(* IEC 61131-3 sources: ST-Study/patterns, 3 files *)

(* ---- fb_alarm_manager.st ---- *)
(*
===============================================================================
  报警管理模块 - FB_AlarmManager
===============================================================================
  功能: 管理多路报警,支持锁存/复位/确认/消抖/优先级
  作者: ST 学习系统
  版本: v1.0
  日期: 2025-12-21

  使用场景:
  - 管理多个报警源(传感器故障、超时、越限等)
  - 需要报警锁存(故障瞬间消失也要记录)
  - 需要报警确认(操作员必须确认才能消除)
  - 需要报警消抖(避免抖动误报)

  核心功能:
  1. 报警锁存: 触发后即使条件消失也保持
  2. 报警复位: 需要人工确认或自动复位
  3. 报警消抖: 信号稳定一段时间才触发
  4. 优先级分类: 严重/警告/提示

  接口说明(单路报警版):
  输入:
    iAlarmTrigger   : BOOL  - 报警触发条件
    iReset          : BOOL  - 复位信号
    iAutoReset      : BOOL  - 允许自动复位
    tDebounceTime   : TIME  - 消抖时间
    nPriority       : INT   - 优先级(1=提示,2=警告,3=严重)

  输出:
    oAlarmActive    : BOOL  - 报警有效(锁存后)
    oAlarmRaw       : BOOL  - 原始报警(消抖后,未锁存)
    oAlarmNew       : BOOL  - 新报警(上升沿脉冲)

  使用示例:
    fbAlarm_MotorOverload(
        iAlarmTrigger := MotorCurrent > MAX_CURRENT,
        iReset := ResetButton,
        iAutoReset := FALSE,  // 严重故障,必须人工复位
        tDebounceTime := T#500ms,
        nPriority := 3,
        oAlarmActive => AlarmLamp
    );
===============================================================================
*)

FUNCTION_BLOCK FB_Alarm
(*
    单路报警模块(基础版)
*)
VAR_INPUT
    iAlarmTrigger   : BOOL;         // 报警触发条件
    iReset          : BOOL;         // 复位信号
    iAutoReset      : BOOL;         // 允许自动复位
    tDebounceTime   : TIME := T#0s; // 消抖时间(0表示不消抖)
    nPriority       : INT := 2;     // 优先级(1=提示,2=警告,3=严重)
END_VAR

VAR_OUTPUT
    oAlarmActive    : BOOL;         // 报警有效(锁存后)
    oAlarmRaw       : BOOL;         // 原始报警(消抖后)
    oAlarmNew       : BOOL;         // 新报警标志(上升沿)
END_VAR

VAR
    fbDebounce      : TON;          // 消抖定时器
    bAlarmLatched   : BOOL;         // 报警锁存
    rtAlarm         : R_TRIG;       // 报警上升沿
    rtReset         : R_TRIG;       // 复位上升沿
END_VAR

// === 消抖处理 ===
fbDebounce(IN := iAlarmTrigger, PT := tDebounceTime);

IF tDebounceTime > T#0s THEN
    oAlarmRaw := fbDebounce.Q;  // 有消抖时间,使用定时器输出
ELSE
    oAlarmRaw := iAlarmTrigger; // 无消抖时间,直接使用原始信号
END_IF

// === 报警锁存 ===
rtAlarm(CLK := oAlarmRaw);
IF rtAlarm.Q THEN
    bAlarmLatched := TRUE;  // 上升沿锁存
END_IF

// === 报警复位 ===
rtReset(CLK := iReset);

// 人工复位
IF rtReset.Q THEN
    bAlarmLatched := FALSE;
END_IF

// 自动复位(条件消失且允许自动复位)
IF iAutoReset AND NOT oAlarmRaw THEN
    bAlarmLatched := FALSE;
END_IF

// === 输出赋值 ===
oAlarmActive := bAlarmLatched;
oAlarmNew := rtAlarm.Q;  // 新报警脉冲(用于计数/记录)

END_FUNCTION_BLOCK

(*
===============================================================================
  多路报警管理器 - FB_AlarmManager
===============================================================================
  管理多路报警(最多16路)
  提供统一的复位、优先级排序、报警计数功能
===============================================================================
*)

FUNCTION_BLOCK FB_AlarmManager

VAR_INPUT
    iAlarmTriggers  : ARRAY[1..16] OF BOOL;  // 16路报警触发条件
    iResetAll       : BOOL;                   // 全部复位
    iResetSingle    : INT;                    // 单路复位(1-16, 0=无)
END_VAR

VAR_OUTPUT
    oAlarmActive    : ARRAY[1..16] OF BOOL;  // 16路报警状态
    oAnyAlarm       : BOOL;                   // 任意报警有效
    oAlarmCount     : INT;                    // 当前报警数量
    oHighestPriority: INT;                    // 最高优先级(3=严重,2=警告,1=提示)
END_VAR

VAR
    fbAlarms        : ARRAY[1..16] OF FB_Alarm;  // 16个报警实例
    i               : INT;                        // 循环变量

    // 每路报警的配置(可外部配置或在此硬编码)
    aPriority       : ARRAY[1..16] OF INT := [
        3, 3, 2, 2, 2, 2, 1, 1,  // 路1-8
        1, 1, 1, 1, 1, 1, 1, 1   // 路9-16
    ];

    aDebounceTime   : ARRAY[1..16] OF TIME := [
        T#500ms, T#500ms, T#300ms, T#300ms, T#300ms, T#300ms, T#200ms, T#200ms,
        T#200ms, T#200ms, T#200ms, T#200ms, T#200ms, T#200ms, T#200ms, T#200ms
    ];

    aAutoReset      : ARRAY[1..16] OF BOOL := [
        FALSE, FALSE, FALSE, FALSE, TRUE, TRUE, TRUE, TRUE,
        TRUE, TRUE, TRUE, TRUE, TRUE, TRUE, TRUE, TRUE
    ];
END_VAR

// === 循环处理每路报警 ===
oAlarmCount := 0;
oHighestPriority := 0;

FOR i := 1 TO 16 DO
    // 调用单路报警模块
    fbAlarms[i](
        iAlarmTrigger := iAlarmTriggers[i],
        iReset := iResetAll OR (iResetSingle = i),
        iAutoReset := aAutoReset[i],
        tDebounceTime := aDebounceTime[i],
        nPriority := aPriority[i],
        oAlarmActive => oAlarmActive[i]
    );

    // 统计报警数量
    IF oAlarmActive[i] THEN
        oAlarmCount := oAlarmCount + 1;

        // 更新最高优先级
        IF aPriority[i] > oHighestPriority THEN
            oHighestPriority := aPriority[i];
        END_IF
    END_IF
END_FOR

// === 任意报警标志 ===
oAnyAlarm := (oAlarmCount > 0);

END_FUNCTION_BLOCK

(*
===============================================================================
  使用示例1: 单路报警
===============================================================================

VAR
    fbAlarm_MotorOverload : FB_Alarm;
    MotorCurrent : REAL;
    MAX_CURRENT : REAL := 10.0;
END_VAR

// 电机过载报警
fbAlarm_MotorOverload(
    iAlarmTrigger := (MotorCurrent > MAX_CURRENT),  // 触发条件
    iReset := HMI.ResetButton,                       // 复位按钮
    iAutoReset := FALSE,                             // 必须人工复位
    tDebounceTime := T#500ms,                        // 消抖500ms
    nPriority := 3,                                  // 严重报警
    oAlarmActive => HMI.AlarmLamp                    // 输出到报警灯
);

// 报警触发时停机
IF fbAlarm_MotorOverload.oAlarmActive THEN
    Motor.iStop := TRUE;
END_IF

===============================================================================
  使用示例2: 多路报警管理
===============================================================================

VAR
    fbAlarmMgr : FB_AlarmManager;

    // 报警触发条件
    bOverload : BOOL;
    bOverheat : BOOL;
    bLowPressure : BOOL;
    // ...
END_VAR

// 配置报警触发条件
fbAlarmMgr.iAlarmTriggers[1] := bOverload;       // 路1: 过载
fbAlarmMgr.iAlarmTriggers[2] := bOverheat;       // 路2: 过热
fbAlarmMgr.iAlarmTriggers[3] := bLowPressure;    // 路3: 低压
// ...

// 调用报警管理器
fbAlarmMgr(
    iResetAll := HMI.ResetAllButton,
    iResetSingle := HMI.SelectedAlarmIndex  // 单个复位
);

// 显示报警状态
HMI.AlarmCount := fbAlarmMgr.oAlarmCount;
HMI.AnyAlarmActive := fbAlarmMgr.oAnyAlarm;

// 根据优先级控制报警灯颜色
CASE fbAlarmMgr.oHighestPriority OF
    3: HMI.AlarmLampColor := RED;     // 严重
    2: HMI.AlarmLampColor := YELLOW;  // 警告
    1: HMI.AlarmLampColor := BLUE;    // 提示
    ELSE
        HMI.AlarmLampColor := OFF;
END_CASE

===============================================================================
  使用示例3: 报警与状态机联动
===============================================================================

FUNCTION_BLOCK FB_MachineControl
VAR
    fbAlarmMgr : FB_AlarmManager;
    nState : INT;
END_VAR

// 严重报警时自动停机
IF fbAlarmMgr.oHighestPriority >= 3 THEN
    nState := STATE_ERROR;  // 进入错误状态
END_IF

// 警告时仅提示,不停机
IF fbAlarmMgr.oHighestPriority = 2 THEN
    HMI.WarningMessage := 'Warning: Check system';
END_IF

END_FUNCTION_BLOCK

===============================================================================
  测试清单
===============================================================================

【基础功能】
1. 触发条件成立 → oAlarmActive=TRUE
2. 触发条件消失,人工复位 → oAlarmActive=FALSE

【锁存机制】
3. 触发条件瞬间成立(100ms)后消失 → oAlarmActive=TRUE(锁存保持)
4. 锁存后必须复位才能消除 → 即使触发条件消失也保持

【消抖功能】
5. 触发条件抖动(ON 100ms, OFF 100ms) → 无报警(未达到消抖时间)
6. 触发条件稳定500ms → 报警触发

【自动复位】
7. 允许自动复位,触发条件消失 → oAlarmActive=FALSE(自动复位)
8. 不允许自动复位,触发条件消失 → oAlarmActive=TRUE(保持,需人工复位)

【多路报警】
9. 3路同时报警 → oAlarmCount=3, oAnyAlarm=TRUE
10. 复位全部 → oAlarmCount=0, oAnyAlarm=FALSE
11. 单个复位路2 → 路2复位,其他保持

【优先级排序】
12. 路1(严重),路3(警告)同时报警 → oHighestPriority=3
13. 路1复位后 → oHighestPriority=2

【边界条件】
14. 连续触发10次 → oAlarmNew只在第一次触发时为TRUE(上升沿)
15. 复位按钮连按10次 → 只复位一次(边沿检测)

===============================================================================
  设计要点
===============================================================================

1. **锁存 vs 非锁存**:
   - 锁存: 故障瞬间即记录,需人工确认(适用于严重故障)
   - 非锁存(自动复位): 条件消失即恢复(适用于轻微提示)

2. **消抖时间选择**:
   - 机械触点: 50-200ms
   - 传感器信号: 100-500ms
   - 模拟量越限: 500-1000ms(避免边界抖动)

3. **优先级分类建议**:
   - 3 严重: 必须立即停机(过载、急停、安全门打开)
   - 2 警告: 需要关注但可继续运行(温度偏高、压力偏低)
   - 1 提示: 仅提示信息(维护提醒、计数达到)

4. **报警历史记录**(扩展):
   - 可添加 ARRAY[1..100] OF AlarmRecord 记录最近100条
   - 记录: 时间戳、报警ID、触发值、复位时间

5. **报警优先级显示**:
   - 严重: 红色闪烁 + 蜂鸣器
   - 警告: 黄色常亮
   - 提示: 蓝色常亮

===============================================================================
*)

(* ---- fb_pause_resume.st ---- *)
(*
===============================================================================
  全局暂停保持模块 - FB_PauseResume
===============================================================================
  功能: 提供全局暂停保持功能,支持多设备同步暂停/恢复
  作者: ST 学习系统
  版本: v1.0
  日期: 2025-12-21

  使用场景:
  - 整条生产线的全局暂停(所有设备同步暂停)
  - 需要保持现场状态的暂停(不是急停,而是"定格")
  - 需要从暂停点精确恢复的场景

  核心思想:
  - 暂停时"冻结"所有状态,不改变任何输出
  - 恢复时从冻结点继续,不重复执行已完成的动作
  - 提供"暂停允许条件"检查,避免危险位置暂停

  接口说明:
  输入:
    iPauseRequest   : BOOL  - 暂停请求
    iResumeRequest  : BOOL  - 恢复请求
    iEmergencyStop  : BOOL  - 急停(强制暂停,不检查条件)
    iPauseEnable    : BOOL  - 暂停允许条件(TRUE时才能暂停)

  输出:
    oPaused         : BOOL  - 当前已暂停
    oPauseActive    : BOOL  - 暂停信号有效(供其他模块读取)
    oResuming       : BOOL  - 恢复中(可用于渐进恢复)
    oPauseRejected  : BOOL  - 暂停请求被拒绝(条件不满足)

  使用示例:
    // 1. 在主程序中实例化(全局单例)
    fbGlobalPause : FB_PauseResume;

    // 2. 调用
    fbGlobalPause(
        iPauseRequest := PauseButton,
        iResumeRequest := ResumeButton,
        iEmergencyStop := EmergencyStop,
        iPauseEnable := SafePositionReached,  // 只在安全位置允许暂停
        oPaused => SystemPaused,
        oPauseActive => GlobalPauseSignal
    );

    // 3. 其他模块响应暂停信号
    IF fbGlobalPause.oPauseActive THEN
        // 冻结当前状态,不改变输出
        RETURN;  // 提前退出,不执行后续逻辑
    END_IF
===============================================================================
*)

FUNCTION_BLOCK FB_PauseResume

VAR_INPUT
    iPauseRequest   : BOOL;     // 暂停请求
    iResumeRequest  : BOOL;     // 恢复请求
    iEmergencyStop  : BOOL;     // 急停信号
    iPauseEnable    : BOOL;     // 暂停允许条件
END_VAR

VAR_OUTPUT
    oPaused         : BOOL;     // 当前已暂停
    oPauseActive    : BOOL;     // 暂停信号有效(供其他模块读取)
    oResuming       : BOOL;     // 恢复中
    oPauseRejected  : BOOL;     // 暂停请求被拒绝
END_VAR

VAR
    bPausedState    : BOOL;     // 暂停状态锁存
    bResumingState  : BOOL;     // 恢复状态

    rtPause         : R_TRIG;   // 暂停上升沿
    rtResume        : R_TRIG;   // 恢复上升沿

    fbRejectPulse   : TP;       // 拒绝脉冲(用于显示)

    CONST_REJECT_PULSE_TIME : TIME := T#2s;  // 拒绝提示持续时间
END_VAR

// === 边沿检测 ===
rtPause(CLK := iPauseRequest);
rtResume(CLK := iResumeRequest);

// === 暂停逻辑 ===
IF rtPause.Q THEN
    // 检查暂停条件
    IF iPauseEnable OR iEmergencyStop THEN
        // 条件满足,执行暂停
        bPausedState := TRUE;
        bResumingState := FALSE;
        oPauseRejected := FALSE;
    ELSE
        // 条件不满足,拒绝暂停
        fbRejectPulse(IN := TRUE, PT := CONST_REJECT_PULSE_TIME);
    END_IF
END_IF

// === 急停强制暂停(优先级最高) ===
IF iEmergencyStop THEN
    bPausedState := TRUE;
    bResumingState := FALSE;
END_IF

// === 恢复逻辑 ===
IF rtResume.Q AND bPausedState AND NOT iEmergencyStop THEN
    bPausedState := FALSE;
    bResumingState := TRUE;  // 进入恢复中状态
END_IF

// === 恢复中状态处理(可用于渐进恢复) ===
IF bResumingState THEN
    // 这里可以添加渐进恢复逻辑
    // 例如:先恢复低速,再恢复正常速度
    // 目前简化为立即恢复
    bResumingState := FALSE;
END_IF

// === 输出赋值 ===
oPaused := bPausedState;
oPauseActive := bPausedState;  // 供其他模块读取的暂停信号
oResuming := bResumingState;

// === 拒绝提示脉冲 ===
fbRejectPulse(IN := FALSE);  // 自动关闭输入
oPauseRejected := fbRejectPulse.Q;

END_FUNCTION_BLOCK

(*
===============================================================================
  使用模式1: 全局暂停(单例模式)
===============================================================================

// === 在全局变量(GVL)中声明 ===
VAR_GLOBAL
    fbGlobalPause : FB_PauseResume;  // 全局唯一实例
END_VAR

// === 在主程序中调用 ===
PROGRAM Main
VAR
    SafePositionReached : BOOL;  // 安全位置标志
END_VAR

// 调用全局暂停模块
fbGlobalPause(
    iPauseRequest := HMI.PauseButton,
    iResumeRequest := HMI.ResumeButton,
    iEmergencyStop := IO.EmergencyStop,
    iPauseEnable := SafePositionReached,  // 只在安全位置允许暂停
    oPaused => HMI.PausedLamp,
    oPauseRejected => HMI.PauseRejectedAlarm
);

// 检查安全位置(示例:所有电机都停止)
SafePositionReached :=
    NOT Motor1.oRunning AND
    NOT Motor2.oRunning AND
    NOT Conveyor.oRunning;

END_PROGRAM

===============================================================================
  使用模式2: 状态机响应全局暂停
===============================================================================

FUNCTION_BLOCK FB_ConveyorControl
VAR_INPUT
    iStart : BOOL;
END_VAR
VAR_OUTPUT
    oRunning : BOOL;
END_VAR
VAR
    nState : INT;
END_VAR

// === 暂停优先检查(在状态机最前面) ===
IF fbGlobalPause.oPauseActive THEN
    // 暂停时冻结状态,不执行后续逻辑
    RETURN;
END_IF

// === 状态机正常逻辑 ===
CASE nState OF
    0: // 空闲
        IF iStart THEN
            nState := 10;
        END_IF

    10: // 启动
        oRunning := TRUE;
        // ...
END_CASE

END_FUNCTION_BLOCK

===============================================================================
  使用模式3: 渐进恢复(高级用法)
===============================================================================

// 修改 FB_PauseResume 的恢复逻辑:
VAR
    fbResumeDelay : TON;  // 恢复延时
    nResumePhase : INT;   // 恢复阶段
END_VAR

// 恢复时分阶段处理
IF rtResume.Q AND bPausedState AND NOT iEmergencyStop THEN
    bPausedState := FALSE;
    bResumingState := TRUE;
    nResumePhase := 1;  // 开始第一阶段
END_IF

IF bResumingState THEN
    CASE nResumePhase OF
        1:  // 第一阶段:低速恢复
            fbResumeDelay(IN := TRUE, PT := T#2s);
            IF fbResumeDelay.Q THEN
                nResumePhase := 2;
                fbResumeDelay(IN := FALSE);
            END_IF

        2:  // 第二阶段:正常速度
            bResumingState := FALSE;
            nResumePhase := 0;
    END_CASE
END_IF

// 其他模块根据 oResuming 调整速度
IF fbGlobalPause.oResuming THEN
    MotorSpeed := LowSpeed;  // 恢复阶段使用低速
ELSE
    MotorSpeed := NormalSpeed;
END_IF

===============================================================================
  测试清单
===============================================================================

【基础功能】
1. 按暂停按钮(条件满足) → oPaused=TRUE, 所有设备冻结
2. 暂停状态按恢复 → oPaused=FALSE, 设备从暂停点继续

【暂停条件检查】
3. 设备运行中按暂停(条件不满足) → oPauseRejected=TRUE, 暂停失败
4. 设备停止后按暂停(条件满足) → oPaused=TRUE, 暂停成功

【急停处理】
5. 运行中急停 → oPaused=TRUE (强制暂停,不检查条件)
6. 急停状态按恢复 → 无效,必须先解除急停

【状态保持】
7. 暂停时传送带位置X → 恢复后仍从位置X继续(不回退)
8. 暂停时计数器值100 → 恢复后从100继续计数(不清零)

【边界条件】
9. 连续按暂停10次 → 只暂停一次(边沿检测)
10. 暂停后立即按恢复 → 正常恢复(无延时限制)
11. 未暂停时按恢复 → 无效(无副作用)

【多设备同步】
12. 3台电机运行,暂停 → 3台同时冻结
13. 恢复 → 3台同时恢复,保持相对位置关系

【拒绝提示】
14. 暂停被拒绝 → oPauseRejected 保持2秒(提示用户)

===============================================================================
  设计要点
===============================================================================

1. **暂停 ≠ 急停**:
   - 暂停: 可控的、可恢复的、保持现场的"定格"
   - 急停: 紧急的、安全的、可能丢失状态的"硬停"

2. **暂停条件检查**:
   - 避免危险位置暂停(如:机械手在空中)
   - 建议: 只在设备停稳、无运动时允许暂停
   - 特殊需求: 可以设计"运动中暂停"(需要额外的位置保存逻辑)

3. **状态冻结技巧**:
   - 在每个FB最前面检查 oPauseActive
   - 如果暂停,RETURN 提前退出,不执行后续逻辑
   - 不改变任何输出,保持现场

4. **恢复策略**:
   - 简单场景: 直接恢复
   - 复杂场景: 渐进恢复(低速→正常速度)
   - 安全场景: 恢复前重新检查安全条件

5. **全局单例模式**:
   - 整个系统只需要一个 FB_PauseResume 实例
   - 在全局变量(GVL)中声明
   - 所有模块读取同一个 oPauseActive 信号

===============================================================================
*)

(* ---- fb_state_machine.st ---- *)
(*
===============================================================================
  通用状态机框架 - FB_StateMachine
===============================================================================
  功能: 提供标准的状态机结构,支持暂停保持/恢复/异常回退
  作者: ST 学习系统
  版本: v1.0
  日期: 2025-12-21

  使用场景:
  - 任何需要步进控制的场景(传送带启动、机械手动作、工序流程等)
  - 需要暂停保持和恢复续跑的自动化流程
  - 需要异常处理和安全回退的控制逻辑

  接口说明:
  输入:
    iStart      : BOOL  - 启动信号(上升沿触发)
    iReset      : BOOL  - 复位信号(回到初始状态)
    iPause      : BOOL  - 暂停信号(保持当前状态)
    iResume     : BOOL  - 恢复信号(从暂停状态继续)
    iEmergency  : BOOL  - 急停信号(立即进入急停状态)

  输出:
    oRunning    : BOOL  - 流程运行中
    oPaused     : BOOL  - 流程已暂停
    oError      : BOOL  - 流程出错
    oComplete   : BOOL  - 流程完成
    nCurrentStep: INT   - 当前步号(用于监控)
    sStepName   : STRING- 当前步名称(用于调试)

  内部变量:
    nState      : INT   - 状态机当前状态
    nStateLast  : INT   - 暂停前的状态(用于恢复)
    bFirstScan  : BOOL  - 每个状态的首次扫描标志

  使用示例:
    fbMachine(
        iStart := StartButton,
        iReset := ResetButton,
        iPause := PauseButton,
        iResume := ResumeButton,
        iEmergency := EmergencyStop,
        oRunning => SystemRunning,
        oPaused => SystemPaused,
        oError => SystemError,
        oComplete => SystemComplete,
        nCurrentStep => CurrentStepDisplay
    );
===============================================================================
*)

FUNCTION_BLOCK FB_StateMachine

VAR_INPUT
    iStart      : BOOL;     // 启动信号
    iReset      : BOOL;     // 复位信号
    iPause      : BOOL;     // 暂停信号
    iResume     : BOOL;     // 恢复信号
    iEmergency  : BOOL;     // 急停信号
END_VAR

VAR_OUTPUT
    oRunning    : BOOL;     // 运行中
    oPaused     : BOOL;     // 已暂停
    oError      : BOOL;     // 出错
    oComplete   : BOOL;     // 完成
    nCurrentStep: INT;      // 当前步号
    sStepName   : STRING;   // 当前步名称
END_VAR

VAR
    nState      : INT := 0;     // 当前状态
    nStateLast  : INT := 0;     // 暂停前状态(用于恢复)
    bFirstScan  : BOOL;         // 首次扫描标志

    // 边沿检测
    rtStart     : R_TRIG;       // 启动上升沿
    rtReset     : R_TRIG;       // 复位上升沿
    rtPause     : R_TRIG;       // 暂停上升沿
    rtResume    : R_TRIG;       // 恢复上升沿
END_VAR

VAR CONSTANT
    // 系统状态定义(负数为特殊状态)
    STATE_IDLE      : INT := 0;     // 空闲
    STATE_PAUSE     : INT := -1;    // 暂停
    STATE_ERROR     : INT := -2;    // 错误
    STATE_EMERGENCY : INT := -3;    // 急停

    // 工作状态定义(根据实际流程修改)
    STATE_INIT      : INT := 1;     // 初始化
    STATE_STEP1     : INT := 10;    // 步骤1
    STATE_STEP2     : INT := 20;    // 步骤2
    STATE_STEP3     : INT := 30;    // 步骤3
    STATE_COMPLETE  : INT := 100;   // 完成
END_VAR

// === 边沿检测 ===
rtStart(CLK := iStart);
rtReset(CLK := iReset);
rtPause(CLK := iPause);
rtResume(CLK := iResume);

// === 急停优先(任何状态下都响应) ===
IF iEmergency THEN
    nState := STATE_EMERGENCY;
    bFirstScan := TRUE;
END_IF

// === 复位处理(次优先) ===
IF rtReset.Q AND NOT iEmergency THEN
    nState := STATE_IDLE;
    bFirstScan := TRUE;
END_IF

// === 暂停/恢复处理 ===
IF rtPause.Q AND nState > 0 THEN  // 只在工作状态下暂停
    nStateLast := nState;         // 保存当前状态
    nState := STATE_PAUSE;
    bFirstScan := TRUE;
END_IF

IF rtResume.Q AND nState = STATE_PAUSE THEN
    nState := nStateLast;         // 恢复到暂停前状态
    bFirstScan := FALSE;          // 恢复时不执行首次扫描动作
END_IF

// === 状态机主逻辑 ===
CASE nState OF

    // -------------------------------------------------------------------------
    // 空闲状态
    // -------------------------------------------------------------------------
    STATE_IDLE:
        sStepName := 'IDLE';
        oRunning := FALSE;
        oPaused := FALSE;
        oError := FALSE;
        oComplete := FALSE;

        // 等待启动信号
        IF rtStart.Q AND NOT iEmergency THEN
            nState := STATE_INIT;
            bFirstScan := TRUE;
        END_IF

    // -------------------------------------------------------------------------
    // 初始化状态
    // -------------------------------------------------------------------------
    STATE_INIT:
        sStepName := 'INIT';
        oRunning := TRUE;
        oComplete := FALSE;

        IF bFirstScan THEN
            // 首次进入该状态时执行的动作
            // TODO: 添加初始化动作(如:复位计数器、清除标志位等)
            bFirstScan := FALSE;
        END_IF

        // TODO: 添加初始化完成条件
        IF TRUE THEN  // 替换为实际完成条件
            nState := STATE_STEP1;
            bFirstScan := TRUE;
        END_IF

    // -------------------------------------------------------------------------
    // 步骤1
    // -------------------------------------------------------------------------
    STATE_STEP1:
        sStepName := 'STEP1';
        oRunning := TRUE;

        IF bFirstScan THEN
            // TODO: 添加步骤1的启动动作
            bFirstScan := FALSE;
        END_IF

        // TODO: 添加步骤1的持续动作

        // TODO: 添加步骤1的完成条件
        IF TRUE THEN  // 替换为实际完成条件
            nState := STATE_STEP2;
            bFirstScan := TRUE;
        END_IF

        // TODO: 添加步骤1的超时/异常检测
        IF FALSE THEN  // 替换为实际异常条件
            nState := STATE_ERROR;
            bFirstScan := TRUE;
        END_IF

    // -------------------------------------------------------------------------
    // 步骤2
    // -------------------------------------------------------------------------
    STATE_STEP2:
        sStepName := 'STEP2';
        oRunning := TRUE;

        IF bFirstScan THEN
            // TODO: 添加步骤2的启动动作
            bFirstScan := FALSE;
        END_IF

        // TODO: 添加步骤2的完成条件
        IF TRUE THEN  // 替换为实际完成条件
            nState := STATE_STEP3;
            bFirstScan := TRUE;
        END_IF

    // -------------------------------------------------------------------------
    // 步骤3
    // -------------------------------------------------------------------------
    STATE_STEP3:
        sStepName := 'STEP3';
        oRunning := TRUE;

        IF bFirstScan THEN
            // TODO: 添加步骤3的启动动作
            bFirstScan := FALSE;
        END_IF

        // TODO: 添加步骤3的完成条件
        IF TRUE THEN  // 替换为实际完成条件
            nState := STATE_COMPLETE;
            bFirstScan := TRUE;
        END_IF

    // -------------------------------------------------------------------------
    // 完成状态
    // -------------------------------------------------------------------------
    STATE_COMPLETE:
        sStepName := 'COMPLETE';
        oRunning := FALSE;
        oComplete := TRUE;

        // 等待复位或重新启动
        // (复位由全局复位处理,这里可以添加自动复位逻辑)

    // -------------------------------------------------------------------------
    // 暂停状态
    // -------------------------------------------------------------------------
    STATE_PAUSE:
        sStepName := 'PAUSED';
        oPaused := TRUE;

        // 暂停时保持所有输出(不改变任何执行机构状态)
        // 等待恢复或复位信号(由全局处理)

    // -------------------------------------------------------------------------
    // 错误状态
    // -------------------------------------------------------------------------
    STATE_ERROR:
        sStepName := 'ERROR';
        oRunning := FALSE;
        oError := TRUE;

        IF bFirstScan THEN
            // TODO: 添加错误处理动作(如:停止所有输出、报警等)
            bFirstScan := FALSE;
        END_IF

        // 只能通过复位退出错误状态

    // -------------------------------------------------------------------------
    // 急停状态
    // -------------------------------------------------------------------------
    STATE_EMERGENCY:
        sStepName := 'EMERGENCY';
        oRunning := FALSE;
        oError := TRUE;

        IF bFirstScan THEN
            // TODO: 添加急停动作(立即停止所有危险动作)
            bFirstScan := FALSE;
        END_IF

        // 急停解除后需要复位才能继续

    // -------------------------------------------------------------------------
    // 未知状态(安全保护)
    // -------------------------------------------------------------------------
    ELSE
        nState := STATE_ERROR;
        bFirstScan := TRUE;

END_CASE

// === 输出当前步号 ===
nCurrentStep := nState;

END_FUNCTION_BLOCK

(*
===============================================================================
  测试清单
===============================================================================

【基础功能】
1. 空闲状态按启动 → 进入初始化 → 依次执行STEP1/2/3 → 完成
2. 完成后按复位 → 回到空闲状态

【暂停保持】
3. STEP2运行中按暂停 → 进入暂停状态,保持当前输出
4. 暂停状态按恢复 → 回到STEP2继续执行

【急停处理】
5. 任意状态按急停 → 立即进入急停状态
6. 急停解除后必须复位才能重新启动

【边界条件】
7. 连续按启动10次 → 只启动一次(边沿检测)
8. 暂停后按复位 → 直接回到空闲(不需要先恢复)
9. 错误状态按启动 → 无效,必须先复位

【状态一致性】
10. 暂停→恢复 → 从暂停点继续,不重复执行首次扫描动作
11. 掉电恢复到STEP2 → 不自动继续,需要人工确认后启动

【异常处理】
12. STEP1出现异常(超时/传感器故障) → 进入错误状态
13. 错误状态按复位 → 回到空闲,需重新检查故障原因

===============================================================================
  使用提示
===============================================================================

1. **状态号规划**:
   - 负数: 特殊状态(暂停/错误/急停)
   - 0: 空闲
   - 1-99: 工作状态(建议每10个数字一个大步骤)
   - 100+: 结束状态

2. **bFirstScan 用途**:
   - 用于区分"单次执行"和"持续执行"
   - 启动动作(如发脉冲)必须在 bFirstScan=TRUE 时执行
   - 持续动作(如保持输出)不检查 bFirstScan

3. **暂停保持机制**:
   - 暂停时 nStateLast 保存当前状态号
   - 恢复时 bFirstScan=FALSE,避免重复执行启动动作
   - 暂停状态下不改变任何输出(保持现场)

4. **扩展建议**:
   - 添加超时检测(每个步骤加 TON 定时器)
   - 添加步骤计时(记录每步耗时)
   - 添加步骤计数器(统计执行次数)
   - 添加步骤历史(记录最近N步的轨迹)

===============================================================================
*)
